PROGRAM Stn053_65_Stn232Divert
VAR
	fbTC: FB_Stn232DivertTC;
	{attribute 'TcLinkToOSO' := '.iPuckPresent   :=  <0,1,0>TIIB[N41S00 (AL1332)]^N41S03 (AL2341)^TxPDO^input byte 0;
								 .iMainBufferFull   :=  <0,1,0>TIIB[N41S00 (AL1332)]^N41S03 (AL2341)^TxPDO^input byte 2;
								 .iDivertMain   :=  <0,1,1>TIIB[N41S00 (AL1332)]^N41S03 (AL2341)^TxPDO^input byte 2;
								 .iDivertSpur   :=  <0,1,1>TIIB[N41S00 (AL1332)]^N41S03 (AL2341)^TxPDO^input byte 0;
								 .oDivertMain   :=  <0,1,0>TIIB[N41S00 (AL1332)]^N41S02 (EX260)^RxPDO^output byte 1;
								 .oDivertSpur   :=  <0,1,1>TIIB[N41S00 (AL1332)]^N41S02 (EX260)^RxPDO^output byte 1;
								 .oStopLower   :=  <0,1,6>TIIB[N41S00 (AL1332)]^N41S02 (EX260)^RxPDO^output byte 0'}

	{attribute 'TcLinkTo' := '.fbRFID.iRawArray[0] := TIIB[N41S00 (AL1332)]^N41S08 (DTI425)^TxPDO^input byte 0;
                             .fbRFID.iRawArray[1] := TIIB[N41S00 (AL1332)]^N41S08 (DTI425)^TxPDO^input byte 1;
                             .fbRFID.iRawArray[2] := TIIB[N41S00 (AL1332)]^N41S08 (DTI425)^TxPDO^input byte 2;
                             .fbRFID.iRawArray[3] := TIIB[N41S00 (AL1332)]^N41S08 (DTI425)^TxPDO^input byte 3;
                             .fbRFID.iRawArray[4] := TIIB[N41S00 (AL1332)]^N41S08 (DTI425)^TxPDO^input byte 4;
                             .fbRFID.iRawArray[5] := TIIB[N41S00 (AL1332)]^N41S08 (DTI425)^TxPDO^input byte 5;
                             .fbRFID.iRawArray[6] := TIIB[N41S00 (AL1332)]^N41S08 (DTI425)^TxPDO^input byte 6;
                             .fbRFID.iRawArray[7] := TIIB[N41S00 (AL1332)]^N41S08 (DTI425)^TxPDO^input byte 7;
                             .fbRFID.iRawArray[8] := TIIB[N41S00 (AL1332)]^N41S08 (DTI425)^TxPDO^input byte 8;
                             .fbRFID.iRawArray[9] := TIIB[N41S00 (AL1332)]^N41S08 (DTI425)^TxPDO^input byte 9;
                             .fbRFID.iRawArray[10] := TIIB[N41S00 (AL1332)]^N41S08 (DTI425)^TxPDO^input byte 10;
                             .fbRFID.iRawArray[11] := TIIB[N41S00 (AL1332)]^N41S08 (DTI425)^TxPDO^input byte 11;
                             .fbRFID.iRawArray[12] := TIIB[N41S00 (AL1332)]^N41S08 (DTI425)^TxPDO^input byte 12;
                             .fbRFID.iRawArray[13] := TIIB[N41S00 (AL1332)]^N41S08 (DTI425)^TxPDO^input byte 13;
                             .fbRFID.iRawArray[14] := TIIB[N41S00 (AL1332)]^N41S08 (DTI425)^TxPDO^input byte 14;
                             .fbRFID.iRawArray[15] := TIIB[N41S00 (AL1332)]^N41S08 (DTI425)^TxPDO^input byte 15;
                             .fbRFID.iRawArray[16] := TIIB[N41S00 (AL1332)]^N41S08 (DTI425)^TxPDO^input byte 16;
                             .fbRFID.iRawArray[17] := TIIB[N41S00 (AL1332)]^N41S08 (DTI425)^TxPDO^input byte 17;
                             .fbRFID.iRawArray[18] := TIIB[N41S00 (AL1332)]^N41S08 (DTI425)^TxPDO^input byte 18;
                             .fbRFID.iRawArray[19] := TIIB[N41S00 (AL1332)]^N41S08 (DTI425)^TxPDO^input byte 19;
                             .fbRFID.iRawArray[20] := TIIB[N41S00 (AL1332)]^N41S08 (DTI425)^TxPDO^input byte 20;
                             .fbRFID.iRawArray[21] := TIIB[N41S00 (AL1332)]^N41S08 (DTI425)^TxPDO^input byte 21;
                             .fbRFID.iRawArray[22] := TIIB[N41S00 (AL1332)]^N41S08 (DTI425)^TxPDO^input byte 22;
                             .fbRFID.iRawArray[23] := TIIB[N41S00 (AL1332)]^N41S08 (DTI425)^TxPDO^input byte 23;
                             .fbRFID.iRawArray[24] := TIIB[N41S00 (AL1332)]^N41S08 (DTI425)^TxPDO^input byte 24;
                             .fbRFID.iRawArray[25] := TIIB[N41S00 (AL1332)]^N41S08 (DTI425)^TxPDO^input byte 25;
                             .fbRFID.iRawArray[26] := TIIB[N41S00 (AL1332)]^N41S08 (DTI425)^TxPDO^input byte 26;
                             .fbRFID.iRawArray[27] := TIIB[N41S00 (AL1332)]^N41S08 (DTI425)^TxPDO^input byte 27;
                             .fbRFID.iRawArray[28] := TIIB[N41S00 (AL1332)]^N41S08 (DTI425)^TxPDO^input byte 28;
                             .fbRFID.iRawArray[29] := TIIB[N41S00 (AL1332)]^N41S08 (DTI425)^TxPDO^input byte 29;
                             .fbRFID.iRawArray[30] := TIIB[N41S00 (AL1332)]^N41S08 (DTI425)^TxPDO^input byte 30;
                             .fbRFID.iRawArray[31] := TIIB[N41S00 (AL1332)]^N41S08 (DTI425)^TxPDO^input byte 31;
							 .fbRFID.oRawArray[0] := TIIB[N41S00 (AL1332)]^N41S08 (DTI425)^RxPDO^output byte 0;
                             .fbRFID.oRawArray[1] := TIIB[N41S00 (AL1332)]^N41S08 (DTI425)^RxPDO^output byte 1;
                             .fbRFID.oRawArray[2] := TIIB[N41S00 (AL1332)]^N41S08 (DTI425)^RxPDO^output byte 2;
                             .fbRFID.oRawArray[3] := TIIB[N41S00 (AL1332)]^N41S08 (DTI425)^RxPDO^output byte 3;
                             .fbRFID.oRawArray[4] := TIIB[N41S00 (AL1332)]^N41S08 (DTI425)^RxPDO^output byte 4;
                             .fbRFID.oRawArray[5] := TIIB[N41S00 (AL1332)]^N41S08 (DTI425)^RxPDO^output byte 5;
                             .fbRFID.oRawArray[6] := TIIB[N41S00 (AL1332)]^N41S08 (DTI425)^RxPDO^output byte 6;
                             .fbRFID.oRawArray[7] := TIIB[N41S00 (AL1332)]^N41S08 (DTI425)^RxPDO^output byte 7;
                             .fbRFID.oRawArray[8] := TIIB[N41S00 (AL1332)]^N41S08 (DTI425)^RxPDO^output byte 8;
                             .fbRFID.oRawArray[9] := TIIB[N41S00 (AL1332)]^N41S08 (DTI425)^RxPDO^output byte 9;
                             .fbRFID.oRawArray[10] := TIIB[N41S00 (AL1332)]^N41S08 (DTI425)^RxPDO^output byte 10;
                             .fbRFID.oRawArray[11] := TIIB[N41S00 (AL1332)]^N41S08 (DTI425)^RxPDO^output byte 11;
                             .fbRFID.oRawArray[12] := TIIB[N41S00 (AL1332)]^N41S08 (DTI425)^RxPDO^output byte 12;
                             .fbRFID.oRawArray[13] := TIIB[N41S00 (AL1332)]^N41S08 (DTI425)^RxPDO^output byte 13;
                             .fbRFID.oRawArray[14] := TIIB[N41S00 (AL1332)]^N41S08 (DTI425)^RxPDO^output byte 14;
                             .fbRFID.oRawArray[15] := TIIB[N41S00 (AL1332)]^N41S08 (DTI425)^RxPDO^output byte 15;
                             .fbRFID.oRawArray[16] := TIIB[N41S00 (AL1332)]^N41S08 (DTI425)^RxPDO^output byte 16;
                             .fbRFID.oRawArray[17] := TIIB[N41S00 (AL1332)]^N41S08 (DTI425)^RxPDO^output byte 17;
                             .fbRFID.oRawArray[18] := TIIB[N41S00 (AL1332)]^N41S08 (DTI425)^RxPDO^output byte 18;
                             .fbRFID.oRawArray[19] := TIIB[N41S00 (AL1332)]^N41S08 (DTI425)^RxPDO^output byte 19;
                             .fbRFID.oRawArray[20] := TIIB[N41S00 (AL1332)]^N41S08 (DTI425)^RxPDO^output byte 20;
                             .fbRFID.oRawArray[21] := TIIB[N41S00 (AL1332)]^N41S08 (DTI425)^RxPDO^output byte 21;
                             .fbRFID.oRawArray[22] := TIIB[N41S00 (AL1332)]^N41S08 (DTI425)^RxPDO^output byte 22;
                             .fbRFID.oRawArray[23] := TIIB[N41S00 (AL1332)]^N41S08 (DTI425)^RxPDO^output byte 23;
                             .fbRFID.oRawArray[24] := TIIB[N41S00 (AL1332)]^N41S08 (DTI425)^RxPDO^output byte 24;
                             .fbRFID.oRawArray[25] := TIIB[N41S00 (AL1332)]^N41S08 (DTI425)^RxPDO^output byte 25;
                             .fbRFID.oRawArray[26] := TIIB[N41S00 (AL1332)]^N41S08 (DTI425)^RxPDO^output byte 26;
                             .fbRFID.oRawArray[27] := TIIB[N41S00 (AL1332)]^N41S08 (DTI425)^RxPDO^output byte 27;
                             .fbRFID.oRawArray[28] := TIIB[N41S00 (AL1332)]^N41S08 (DTI425)^RxPDO^output byte 28;
                             .fbRFID.oRawArray[29] := TIIB[N41S00 (AL1332)]^N41S08 (DTI425)^RxPDO^output byte 29;
                             .fbRFID.oRawArray[30] := TIIB[N41S00 (AL1332)]^N41S08 (DTI425)^RxPDO^output byte 30;
                             .fbRFID.oRawArray[31] := TIIB[N41S00 (AL1332)]^N41S08 (DTI425)^RxPDO^output byte 31'}
	fbConvDivert: FB_ConvDivertPuck;
	
	Debug_config_IsCRTC1: BOOL := 1;
	Debug_config_IsPilot: BOOL := 0;
	
	Debug_InBypassThisStn: BOOL := 0;
	Debug_InBypassDownstreamStn: BOOL := 0;
	
END_VAR

// Mappings to/from remote stations
gStn053_65_Stn232Divert.MainHeartbeatOK := TRUE; // because this PLC is Main
gStn053_65_Stn232Divert.MainConvRunning :=  gConsumed_SafetyInterfaceConv.MtrRunning.Enc057Mtr01;
gStn053_65_Stn232Divert.MainInAuto := gStn053.CycleAuto;

gStn053_65_Stn232Divert.SpurHeartbeatOK := gConsumed_Stn232To053_OK;
gStn053_65_Stn232Divert.SpurConvRunning := gConsumed_Stn232To053.SpurConvRunning;
gStn053_65_Stn232Divert.SpurInAuto := gConsumed_Stn232To053.StationInAuto;
gStn053_65_Stn232Divert.SpurEmptyRequest := gConsumed_Stn232To053.ScratchPad[0].0;
gStn053_65_Stn232Divert.SpurPurgeMode := gConsumed_Stn232To053.ScratchPad[0].1;
gStn053_65_Stn232Divert.SpurBufferFull := gConsumed_Stn232To053.DivertSpurDSBufferFull;

//TODO RCC - Eventually populate station bypass inputs to TC
// Call to traffic control function block.
fbTC(
	pCmp := ADR(gStn053_65_Stn232Divert)
);

// Call to divert component logic instance.
fbConvDivert(
	pStn := ADR(gStn053),
	pCmp := ADR(gStn053_65_Stn232Divert),
	pStateTraceBuffer := ADR(gStn053_StateTraceBuffer),
	pStateTraceFifo := ADR(gStn053_StateTraceFifo),
	pStats := ADR(gStn053_02_Stats));

END_PROGRAM

(* stored: Version 1.1.0.1, ProductVersion 3.1.4024.6
   POU Stn053_65_Stn232Divert: Id {f24535f8-8f2a-406e-b765-9a81761eb132}, SpecialFunc None *)
